// TIA Portal V20 export
DATA_BLOCK "LBP_TMLoad"   // DB71
TITLE = Tool management / Gestion des outils
{ S7_Optimized_Access := 'FALSE' }
AUTHOR : SINUMERIK
FAMILY : SINUMERIK_ONE
VERSION : 6.24
// Interface between user program and tool management, contains signals from/to Load/Unload magazine / Interface entre programme utilisateur et gestion d'outil, contient des signaux de/vers Chargement/déchargement de magasin
// stored: AutoNumber false, InstanceOfName LBP_typeTMLoad, InstanceOfType UDT
"LBP_typeTMLoad"
   // VAR RETAIN
   //    IFNo : Array[1..16] of Bool;
   //    Quit : Array[1..16] of Bool;
   //    TIF : Array[1..16] of Struct
   //       Loading : Bool;
   //       Unloading : Bool;
   //       Reloading : Bool;
   //       Positioning : Bool;
   //       PosbyProgram : Bool;
   //       PositioningMT : Bool;
   //       f0_6 : Bool;
   //       f0_7 : Bool;
   //       PerfStatusError : Bool;
   //       n1_1 : Bool;
   //       n1_2 : Bool;
   //       n1_3 : Bool;
   //       n1_4 : Bool;
   //       n1_5 : Bool;
   //       n1_6 : Bool;
   //       DataInDB1071 : Bool;
   //       Channel : Byte;
   //       TMNo : Byte;
   //       reserved1 : DInt;
   //       reserved2 : DInt;
   //       reserved3 : DInt;
   //       LoadIdent : Int;
   //       LoadNo : Int;
   //       SMag : Int;
   //       SLoc : Int;
   //       TMag : Int;
   //       TLoc : Int;
   //       WithoutMagMoving : Bool;
   //       Res2 : Byte;
   //    END_STRUCT;
   // END_VAR
BEGIN
END_DATA_BLOCK
